# EPICS autosave request: ADApp/Db/NDOverlay_settings.req
$(P)$(R)Name
$(P)$(R)Use
$(P)$(R)PositionXLink
$(P)$(R)PositionX
$(P)$(R)PositionYLink
$(P)$(R)PositionY
$(P)$(R)SizeXLink
$(P)$(R)SizeX
$(P)$(R)SizeYLink
$(P)$(R)SizeY
$(P)$(R)DrawMode
$(P)$(R)Shape
$(P)$(R)Red
$(P)$(R)Green
$(P)$(R)Blue
